(* CODESYS project Interfaces.export

Project tree, tasks and I/O mapping:
  Interfaces/
    interface itfPreAction: PreAction
*)

// Interfaces/itfPreAction
INTERFACE itfPreAction

METHOD PreAction : bool
VAR_INPUT
END_VAR
END_METHOD

END_INTERFACE
